(* PLC project Thuis, Unknown Unnamed 1 *)
(* stored: creationDateTime 2022-12-23T16:48:11, modificationDateTime 2023-05-13T14:44:54 *)

PROGRAM program0
  VAR
    A5 AT %IX0.0 : BOOL;
    A6 AT %IX0.1 : BOOL;
    A7 AT %IX0.2 : BOOL;
    A8 AT %IX0.3 : BOOL;
    A9 AT %IX0.4 : BOOL;
    A10 AT %IX0.5 : BOOL;
    A11 AT %IX0.6 : BOOL;
    A12 AT %IX0.7 : BOOL;
    A13 AT %IX1.0 : BOOL;
    A14 AT %IX1.1 : BOOL;
    A15 AT %IX1.2 : BOOL;
    I16 AT %IX1.3 : BOOL;
    I17 AT %IX1.4 : BOOL;
    I18 AT %IX1.5 : BOOL;
    IN0 AT %IX1.6 : BOOL;
    IN1 AT %IX1.7 : BOOL;
    R0 AT %QX0.0 : BOOL;
    R1 AT %QX0.1 : BOOL;
    R2 AT %QX0.2 : BOOL;
    R3 AT %QX0.3 : BOOL;
    R4 AT %QX0.4 : BOOL;
    R5 AT %QX0.5 : BOOL;
    R6 AT %QX0.6 : BOOL;
    R7 AT %QX0.7 : BOOL;
    R8 AT %QX1.0 : BOOL;
    R9 AT %QX1.1 : BOOL;
    R10 AT %QX1.2 : BOOL;
    R11 AT %QX1.3 : BOOL;
    R12 AT %QX1.4 : BOOL;
    R13 AT %QX1.5 : BOOL;
    R14 AT %QX1.6 : BOOL;
    R15 AT %QX1.7 : BOOL;
    D0 AT %QX2.0 : BOOL;
    D1 AT %QX2.1 : BOOL;
    D2 AT %QX2.2 : BOOL;
    D3 AT %QX2.3 : BOOL;
    D4 AT %QX2.4 : BOOL;
    D5 AT %QX2.5 : BOOL;
    D6 AT %QX2.6 : BOOL;
    D7 AT %QX2.7 : BOOL;
    D8 AT %QX3.0 : BOOL;
    D9 AT %QX3.1 : BOOL;
    D10 AT %QX3.2 : BOOL;
    D11 AT %QX3.3 : BOOL;
    D12 AT %QX3.4 : BOOL;
    D13 AT %QX3.5 : BOOL;
    D14 AT %QX3.6 : BOOL;
    D15 AT %QX3.7 : BOOL;
    D16 AT %QW0 : UINT;
    ModIn_0 AT %QW1 : WORD;  (* holding register for dimmer *)
    A0 AT %IW0 : WORD;
    A1 AT %IW1 : WORD;
    A2 AT %IW2 : WORD;
    A3 AT %IW3 : WORD;
    A4 AT %IW4 : WORD;
    lumen AT %IW5 : WORD;
  END_VAR

(* FBD diagram, written out as Structured Text *)
END_PROGRAM

(* Impulse relay with central + group on/off *)
FUNCTION_BLOCK Impulse
  VAR_INPUT
    IN : BOOL;  (* Ingang drukknop *)
    GR_ON : BOOL;  (* Groep aan *)
    GR_OFF : BOOL;  (* Groep uit *)
    ALL_ON : BOOL;  (* Alles aan *)
    ALL_OFF : BOOL;  (* Alles uit *)
  END_VAR
  VAR_OUTPUT
    OUT : BOOL;  (* Uitgang relais *)
  END_VAR
  VAR
    SR0 : SR;
    R_TRIG0 : R_TRIG;
  END_VAR

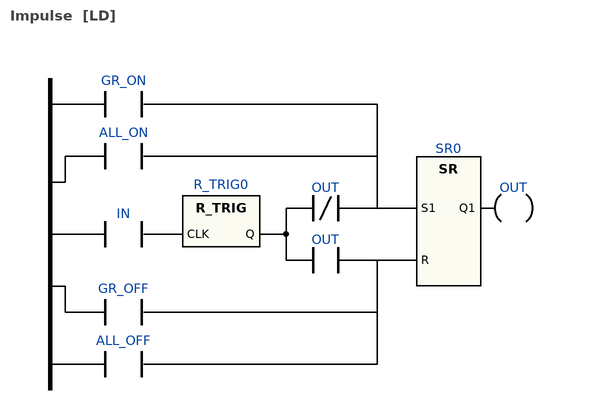
(* LD diagram, written out as Structured Text *)
R_TRIG0(CLK := IN);
SR0(S1 := R_TRIG0.Q AND NOT OUT OR GR_ON OR ALL_ON, R := R_TRIG0.Q AND OUT OR GR_OFF OR ALL_OFF);
OUT := SR0.Q1;
END_FUNCTION_BLOCK

(* Extended Pulse Timer( (re)starts on a pulse) *)
FUNCTION_BLOCK TEP
  VAR_INPUT
    IN : BOOL;
  END_VAR
  VAR_OUTPUT
    Q : BOOL;
  END_VAR
  VAR_INPUT
    PT : TIME;
  END_VAR
  VAR_OUTPUT
    ET : TIME := T#0s;
  END_VAR
  VAR
    STATE : SINT := 0;
    PREV_IN : BOOL := false;
    CURRENT_TIME : TIME;
    START_TIME : TIME;
  END_VAR

              {__SET_VAR(data__->,CURRENT_TIME,,__CURRENT_TIME)}

  IF ((STATE = 0) AND NOT(PREV_IN) AND IN)   (* found rising edge on IN *)
  THEN
    (* start timer... *)
    STATE := 1;
    Q := TRUE;
    START_TIME := CURRENT_TIME;

  ELSIF (STATE = 1)
  THEN
    IF ((START_TIME + PT) <= CURRENT_TIME)
    THEN
      STATE := 2;
      Q := FALSE;
      ET := PT;
    ELSE
      ET := CURRENT_TIME - START_TIME;
    END_IF;
  END_IF;

  IF ((STATE = 2) AND NOT(IN))
  THEN
    ET := T#0s;
    STATE := 0;
  END_IF;


  PREV_IN := IN;
          
END_FUNCTION_BLOCK

(* Short press => Q1 active, long press => Q2 active *)
FUNCTION_BLOCK LenghtOfInputPulse
  VAR_OUTPUT
    Q1 : BOOL;  (* Short press output *)
    Q2 : BOOL;  (* Long press output *)
  END_VAR
  VAR_INPUT
    IN : BOOL;
  END_VAR
  VAR
    TON0 : TON;
    F_TRIG0 : F_TRIG;
  END_VAR

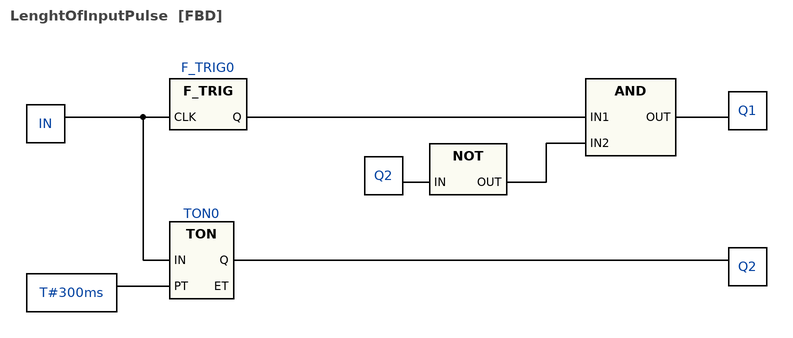
(* FBD diagram, written out as Structured Text *)
F_TRIG0(CLK := IN);
Q1 := F_TRIG0.Q AND NOT Q2;
TON0(IN := IN, PT := T#300ms);
Q2 := TON0.Q;
END_FUNCTION_BLOCK

(* set brightness according to cie1931 *)
FUNCTION_BLOCK LedValue
  VAR_INPUT
    IN : INT;
  END_VAR
  VAR_OUTPUT
    OUT : UINT;
  END_VAR
  VAR
    Values : ARRAY[0..99] OF UINT;
  END_VAR

            Values[ 0 ] := 0;
Values[ 1 ] := 73;
Values[ 2 ] := 147;
Values[ 3 ] := 220;
Values[ 4 ] := 293;
Values[ 5 ] := 366;
Values[ 6 ] := 440;
Values[ 7 ] := 513;
Values[ 8 ] := 586;
Values[ 9 ] := 663;
Values[ 10 ] := 747;
Values[ 11 ] := 837;
Values[ 12 ] := 934;
Values[ 13 ] := 1038;
Values[ 14 ] := 1150;
Values[ 15 ] := 1269;
Values[ 16 ] := 1397;
Values[ 17 ] := 1533;
Values[ 18 ] := 1677;
Values[ 19 ] := 1830;
Values[ 20 ] := 1992;
Values[ 21 ] := 2163;
Values[ 22 ] := 2344;
Values[ 23 ] := 2535;
Values[ 24 ] := 2736;
Values[ 25 ] := 2947;
Values[ 26 ] := 3169;
Values[ 27 ] := 3402;
Values[ 28 ] := 3646;
Values[ 29 ] := 3901;
Values[ 30 ] := 4168;
Values[ 31 ] := 4447;
Values[ 32 ] := 4738;
Values[ 33 ] := 5041;
Values[ 34 ] := 5357;
Values[ 35 ] := 5686;
Values[ 36 ] := 6028;
Values[ 37 ] := 6384;
Values[ 38 ] := 6753;
Values[ 39 ] := 7137;
Values[ 40 ] := 7534;
Values[ 41 ] := 7946;
Values[ 42 ] := 8373;
Values[ 43 ] := 8815;
Values[ 44 ] := 9272;
Values[ 45 ] := 9745;
Values[ 46 ] := 10233;
Values[ 47 ] := 10737;
Values[ 48 ] := 11258;
Values[ 49 ] := 11796;
Values[ 50 ] := 12350;
Values[ 51 ] := 12921;
Values[ 52 ] := 13510;
Values[ 53 ] := 14116;
Values[ 54 ] := 14740;
Values[ 55 ] := 15383;
Values[ 56 ] := 16043;
Values[ 57 ] := 16723;
Values[ 58 ] := 17421;
Values[ 59 ] := 18138;
Values[ 60 ] := 18875;
Values[ 61 ] := 19632;
Values[ 62 ] := 20408;
Values[ 63 ] := 21205;
Values[ 64 ] := 22022;
Values[ 65 ] := 22860;
Values[ 66 ] := 23719;
Values[ 67 ] := 24599;
Values[ 68 ] := 25500;
Values[ 69 ] := 26424;
Values[ 70 ] := 27369;
Values[ 71 ] := 28337;
Values[ 72 ] := 29327;
Values[ 73 ] := 30340;
Values[ 74 ] := 31376;
Values[ 75 ] := 32436;
Values[ 76 ] := 33519;
Values[ 77 ] := 34626;
Values[ 78 ] := 35757;
Values[ 79 ] := 36912;
Values[ 80 ] := 38092;
Values[ 81 ] := 39297;
Values[ 82 ] := 40527;
Values[ 83 ] := 41782;
Values[ 84 ] := 43063;
Values[ 85 ] := 44370;
Values[ 86 ] := 45703;
Values[ 87 ] := 47063;
Values[ 88 ] := 48449;
Values[ 89 ] := 49863;
Values[ 90 ] := 51303;
Values[ 91 ] := 52771;
Values[ 92 ] := 54267;
Values[ 93 ] := 55790;
Values[ 94 ] := 57342;
Values[ 95 ] := 58923;
Values[ 96 ] := 60532;
Values[ 97 ] := 62170;
Values[ 98 ] := 63838;
Values[ 99 ] := 65535;

OUT := Values[ IN ]; 
          
END_FUNCTION_BLOCK

(* Dimmer using a single input. Short pulse, toggle output. Long pulse, dim up/down *)
FUNCTION_BLOCK Dimmer
  VAR_INPUT
    IN : BOOL;  (* input *)
  END_VAR
  VAR_OUTPUT
    OUT : UINT;  (* dimmer output *)
  END_VAR
  VAR_INPUT
    IN_U : BOOL;  (* count up *)
    IN_D : BOOL;  (* count down *)
    GR_ON : BOOL;  (* group on *)
    GR_OFF : BOOL;  (* group off *)
    All_ON : BOOL;  (* all on *)
    All_OFF : BOOL;  (* all off *)
  END_VAR
  VAR
    SR2 : SR;
    PulseLenght : LenghtOfInputPulse;
    Counter : CTUD;
    PT : BOOL := 0;  (* pulse train *)
    StartBit : BOOL := 1;
    SR0 : SR;
    LedValue0 : LedValue;
  END_VAR
  VAR  (* added by the conversion: wires and edge detectors of the diagram *)
    R_TRIG1 : R_TRIG;
    R_TRIG2 : R_TRIG;
  END_VAR

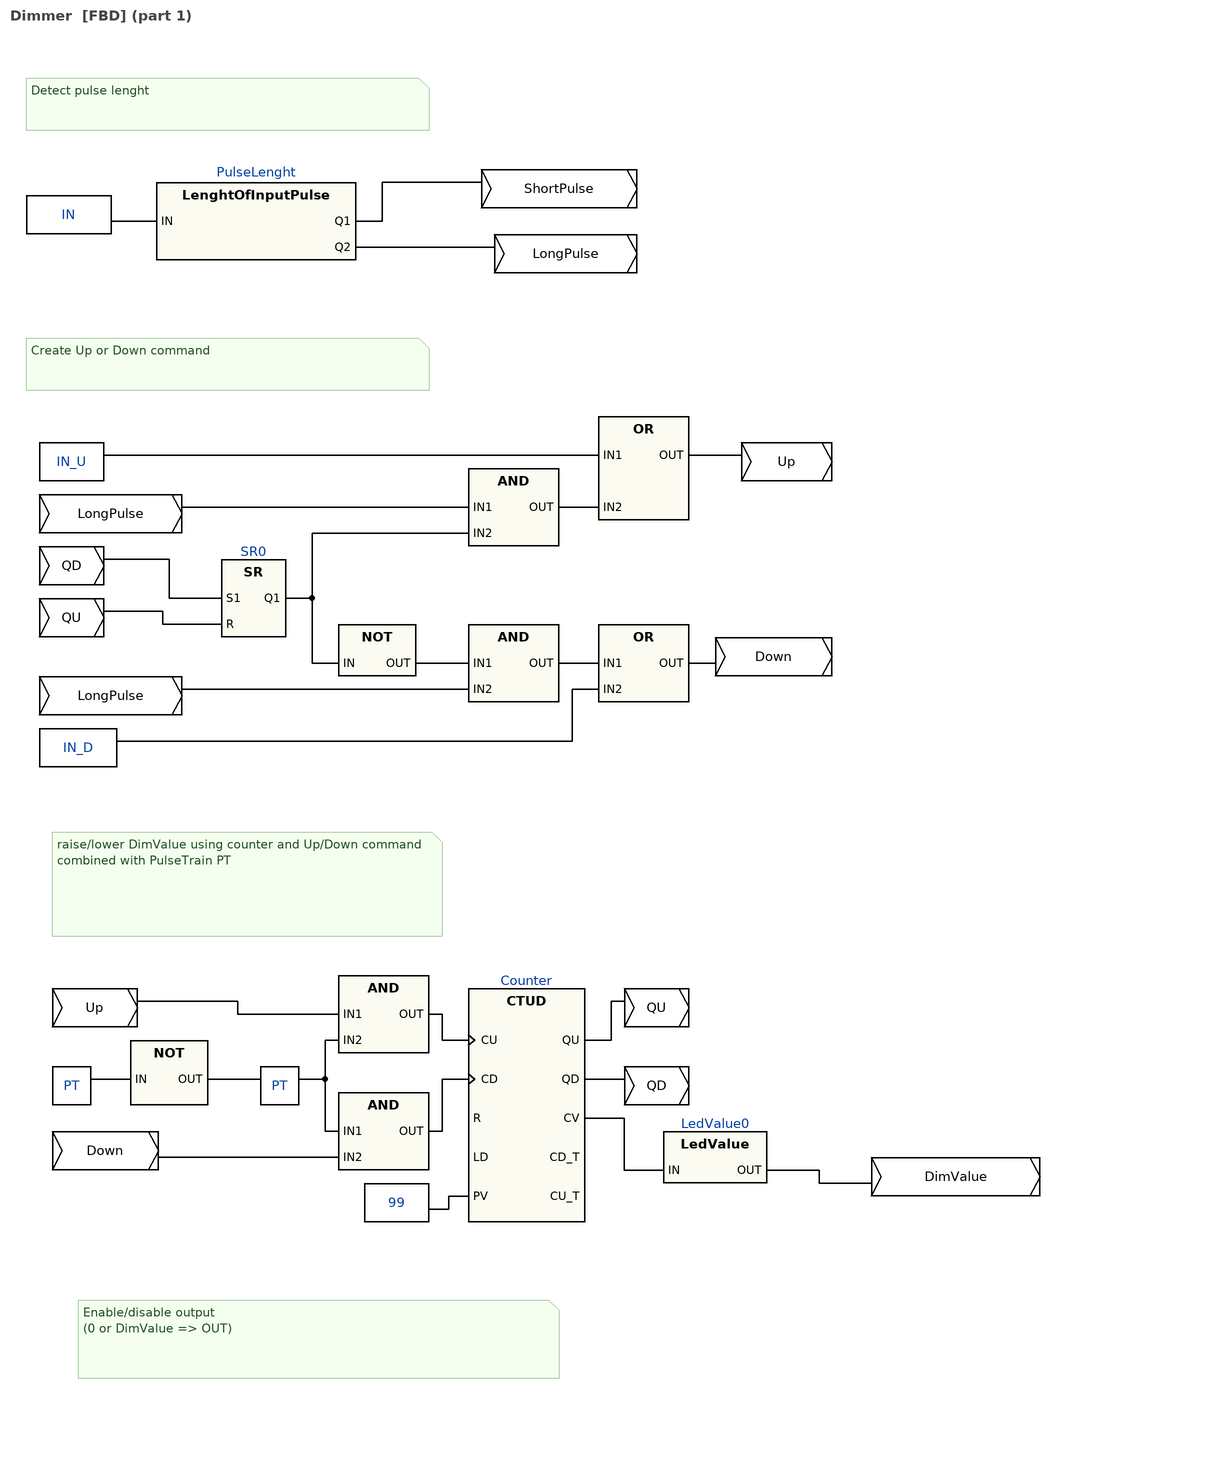
(* FBD diagram, written out as Structured Text *)
(* Detect pulse lenght *)
(* Create Up or Down command *)
(* raise/lower DimValue using counter and Up/Down command combined with PulseTrain PT *)
PT := NOT PT;
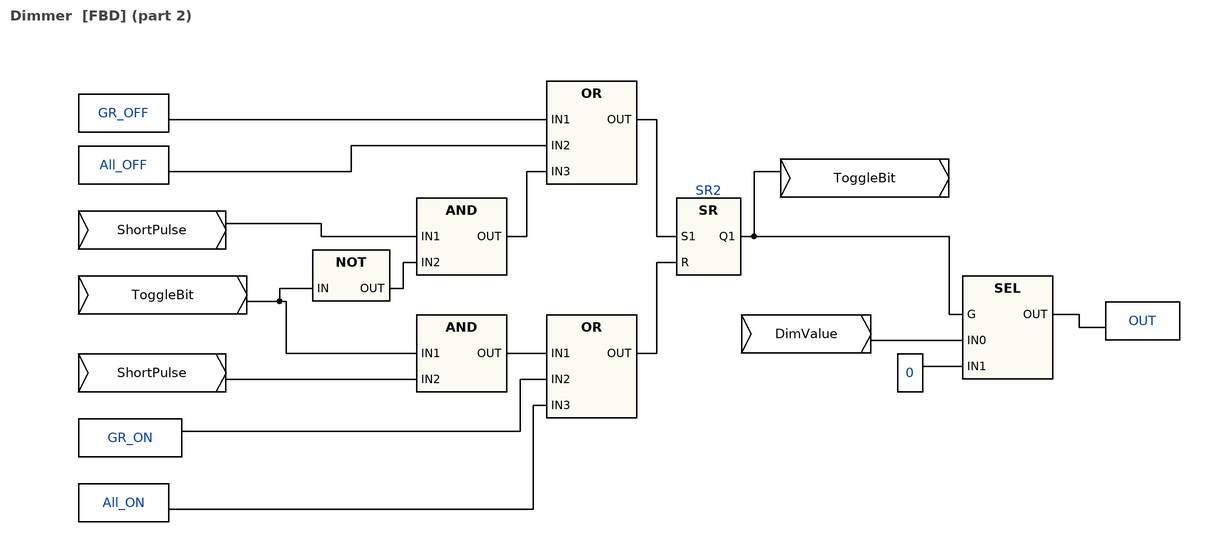
(* Enable/disable output
(0 or DimValue => OUT) *)
PulseLenght(IN := IN);
SR2(S1 := GR_OFF OR All_OFF OR PulseLenght.Q1 AND NOT SR2.Q1, R := SR2.Q1 AND PulseLenght.Q1 OR GR_ON OR All_ON);
SR0(S1 := Counter.QD, R := Counter.QU);
R_TRIG1(CLK := (IN_U OR PulseLenght.Q2 AND SR0.Q1) AND PT);
R_TRIG2(CLK := PT AND (NOT SR0.Q1 AND PulseLenght.Q2 OR IN_D));
Counter(CU := R_TRIG1.Q, CD := R_TRIG2.Q, PV := 99);
LedValue0(IN := Counter.CV);
OUT := SEL(SR2.Q1, LedValue0.OUT, 0);
END_FUNCTION_BLOCK

(* Impulse relay with central + group on/off. Output switches off if longer on as set time. *)
FUNCTION_BLOCK Impulse_t
  VAR_INPUT
    IN : BOOL;
    GR_ON : BOOL;
    GR_OFF : BOOL;
    ALL_ON : BOOL;
    ALL_OFF : BOOL;
    PT : TIME;
  END_VAR
  VAR_OUTPUT
    OUT : BOOL;
  END_VAR
  VAR
    TON0 : TON;
    Impulse0 : Impulse;
  END_VAR

(* FBD diagram, written out as Structured Text *)
TON0(IN := Impulse0.OUT, PT := PT);
Impulse0(IN := IN OR TON0.Q, GR_ON := GR_ON, GR_OFF := GR_OFF, ALL_ON := ALL_ON, ALL_OFF := ALL_OFF);
OUT := Impulse0.OUT;
END_FUNCTION_BLOCK

FUNCTION_BLOCK WordToBit
  VAR_INPUT
    IN : WORD;
  END_VAR
  VAR_OUTPUT
    OUT0 : BOOL;
    OUT1 : BOOL;
    OUT2 : BOOL;
    OUT3 : BOOL;
    OUT4 : BOOL;
    OUT5 : BOOL;
    OUT6 : BOOL;
    OUT7 : BOOL;
    OUT8 : BOOL;
    OUT9 : BOOL;
    OUT10 : BOOL;
    OUT11 : BOOL;
    OUT12 : BOOL;
    OUT13 : BOOL;
    OUT14 : BOOL;
    OUT15 : BOOL;
  END_VAR

            OUT0 := (IN & 1)>0;
OUT1 := (IN & 2)>0;
OUT2 := (IN & 4)>0;
OUT3 := (IN & 8)>0;
OUT4 := (IN & 16)>0;
OUT5 := (IN & 32)>0;
OUT6 := (IN & 64)>0;
OUT7 := (IN & 128)>0;
OUT8 := (IN & 256)>0;
OUT9 := (IN & 512)>0;
OUT10 := (IN & 1024)>0;
OUT11 := (IN & 2048)>0;
OUT12 := (IN & 4096)>0;
OUT13 := (IN & 8192)>0;
OUT14 := (IN & 16384)>0;
OUT15 := (IN & 32768)>0;

          
END_FUNCTION_BLOCK

CONFIGURATION Config0
  RESOURCE Res0 ON PLC
    TASK task0(INTERVAL := T#20ms, PRIORITY := 0);
    PROGRAM instance0 WITH task0 : program0;
  END_RESOURCE
END_CONFIGURATION
